SUBAPPLICATION Uebung_010f3_AX (* SoftKey_F1 ODER AuxFunction2_X1 auf DigitalOutput_Q1 mit GreenWhiteBackground (SoftKey UND Aux) *)
  (* Standard: 61499-2; Description: Copyright (c) 2026 Meisterschulen am Ostbahnhof This program and the accompanying materials are made available under the terms of the Eclipse Public License 2.0 which is available at https://www.eclipse.org/legal/epl-2.0/ SPDX-License-Identifier: EPL-2.0 *)
  (* Version 1.0, 2026-09-06, Franz Höpfinger, Meisterschulen am Ostbahnhof, initial API and implementation and/or initial documentation *)
  PACKAGE Uebungen;
  IMPORT Uebungen::const::UT::DefaultPool::SoftKey_F1;
  IMPORT Uebungen::const::UT::DefaultPool::AuxFunction2_X1;
  IMPORT logiBUS::io::DQ::logiBUS_DO::Output_Q1;
  (* Documentation:
  SoftKey_F1 ODER AuxFunction2_X1 auf DigitalOutput_Q1 mit GreenWhiteBackground
   Kombiniert Uebung_010c_AX (SoftKey mit Background) und Uebung_010f_AX (Aux mit Background) auf einen gemeinsamen Ausgang: dieselbe Funktion ist sowohl über den VT-SoftKey als auch über den physischen Aux-Taster/Joystick bedienbar.
   Funktionsbeschreibung
    - SoftKey_F1 und AuxFunction2_X1 liefern je ein boolesches AX-Signal, AX_OR_2 verknüpft beide per ODER zu einem gemeinsamen Signal für DigitalOutput_Q1.
   - AX_SPLIT_2 verteilt dieses eine Signal auf zwei Ziele: den Ausgang selbst sowie die kombinierte Hintergrundfarbe beider Bedienelemente.
   - GreenWhiteBackground3_AX statt zwei einzelner GreenWhiteBackground1_AX/GreenWhiteBackground2_AX: dieser Baustein nimmt genau einen normalen VT-Objekt-Parameter (u16ObjId = SoftKey) UND einen Aux-Objekt-Parameter (u16ObjIdA = Aux) entgegen und setzt beide Hintergründe aus einem einzigen DI1-Eingang - intern sendet er drei Kommandos (Q_BackgroundColour für den SoftKey, Q_BackgroundColour UND Q_BackgroundColourAux für die Aux-Funktion), aber nach außen genügt ein Split auf zwei statt drei Ziele.
    Arbeitsauftrag
   Testen Sie: SoftKey_F1 drücken → Q1 EIN, beide Hintergründe (SoftKey und Aux) werden grün. Aux-Taster drücken → dasselbe. Werden beide gleichzeitig gehalten, bleibt Q1 EIN, bis beide losgelassen sind - Q1 schaltet erst AUS, wenn sowohl SoftKey_F1 als auch AuxFunction2_X1 wieder FALSE sind (reine ODER-Verknüpfung, kein Latch).
  *)
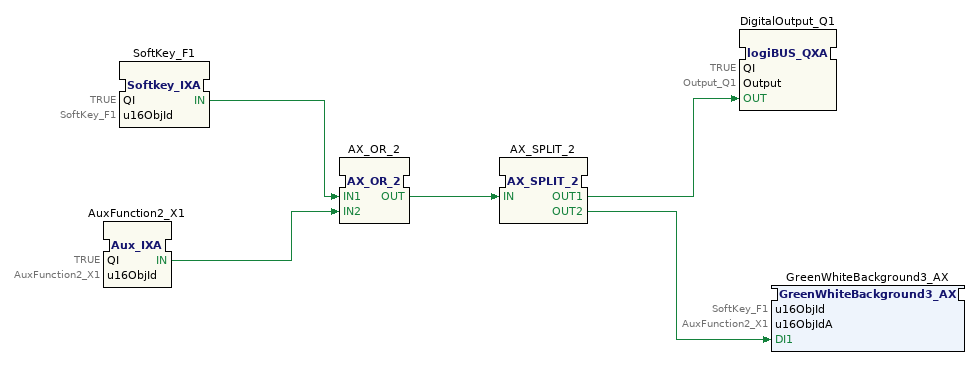
  (* SoftKey_F1 (VT) und AuxFunction2_X1 (Joystick) steuern denselben Q1 - ODER-verknuepft ueber AX_OR_2. GreenWhiteBackground3_AX (nicht 1_AX/2_AX einzeln!) bedient beide Hintergruende aus einem Baustein: u16ObjId=SoftKey (VT) und u16ObjIdA=Aux (VT+Aux-Handle) - siehe Uebung_010f_AX. *)
  FBS
    DigitalOutput_Q1 : logiBUS::io::DQ::logiBUS_QXA(QI := TRUE, Output := Output_Q1);
    SoftKey_F1 : isobus::UT::io::Softkey::Softkey_IXA(QI := TRUE, u16ObjId := SoftKey_F1);
    AuxFunction2_X1 : isobus::UT::io::Auxiliary::IN::Aux_IXA(QI := TRUE, u16ObjId := AuxFunction2_X1);
    AX_OR_2 : adapter::booleanOperators::AX_OR_2;
    AX_SPLIT_2 : adapter::events::unidirectional::AX_SPLIT_2;
  END_FBS
  SUBAPPS
    GreenWhiteBackground3_AX : MyLib::sys::GreenWhiteBackground3_AX(u16ObjId := SoftKey_F1, u16ObjIdA := AuxFunction2_X1);
  END_SUBAPPS
  ADAPTER_CONNECTIONS
    SoftKey_F1.IN TO AX_OR_2.IN1;
    AuxFunction2_X1.IN TO AX_OR_2.IN2;
    AX_OR_2.OUT TO AX_SPLIT_2.IN;
    AX_SPLIT_2.OUT1 TO DigitalOutput_Q1.OUT;
    AX_SPLIT_2.OUT2 TO GreenWhiteBackground3_AX.DI1;
  END_CONNECTIONS
END_SUBAPPLICATION
